FUNCTION_BLOCK FB_LamparaComputada_ST
VAR_INPUT
    ReiniciaContador: BOOL;
    ManiobrasTotales: UINT := 2;
    TiempoEncendido: REAL := 2.0;
END_VAR
VAR_OUTPUT
    LamparaHabilitada: BOOL;
    ManiobrasPendientes: UINT;
    TiempoPendiente: REAL;
END_VAR
VAR
    Lampara AT %Q*: BOOL;
    Pulsador AT %I*: BOOL;
    
    Contador: CTD := (CV := ManiobrasTotales);
    Temporizador: TON;
END_VAR

LamparaHabilitada := NOT Contador.Q;

Contador(
    CD := Lampara,
    LOAD := ReiniciaContador,
    PV := ManiobrasTotales,
    CV => ManiobrasPendientes,
    );

Temporizador(
    IN := Lampara, 
    PT := REAL_TO_TIME(TiempoEncendido * 1000)
    );

IF (LamparaHabilitada AND Pulsador) THEN
    Lampara := TRUE;
ELSIF Temporizador.Q THEN
    Lampara := FALSE;
END_IF

TiempoPendiente := TiempoEncendido - (TIME_TO_REAL(Temporizador.ET) / 1000);

END_FUNCTION_BLOCK

(* stored: Version 1.1.0.1, ProductVersion 3.1.4024.15
   POU FB_LamparaComputada_ST: Id {2c52e490-02c0-48e6-8c38-6edb0e27b45e}, SpecialFunc None *)
